# EPICS autosave request: iocBoot/ioc2/dbSave/23i_KB_Vy_.req
%
% BURT Request File
%
% 23i:KB:Vy:  Vertical KB mirror Y-positioning
%

file $(DIR)/assy.req ASSY=23i:KB:Vy
23i:KB:Vy:BaseLength
file $(DIR)/mtr1.req MTR1=23i:KB:mvy1
file $(DIR)/mtr1.req MTR1=23i:KB:mvy2
file $(DIR)/drv1.req DRV1=23i:KB:VY1
file $(DIR)/drv1.req DRV1=23i:KB:VY2
file $(DIR)/axs1.req AXS1=23i:KB:VL
file $(DIR)/axs1.req AXS1=23i:KB:VW
